// TwinCAT 3 PLC project CPCDAQ_Standard
// ProgramVersion: 3.1.4024.0
// libraries:
//   Tc2_Standard, * (Beckhoff Automation GmbH)
//   Tc2_System, * (Beckhoff Automation GmbH)
//   Tc3_Module, * (Beckhoff Automation GmbH)
// project tree:
//   GVLs/ GVL.TcGVL
//   / PlcTask.TcTTO
//   POUs/ MAIN.TcPOU, POU.TcPOU

CONFIGURATION CPCDAQ_Standard
    RESOURCE PLC ON TwinCAT3
        TASK PlcTask(INTERVAL := T#10ms, PRIORITY := 20);
        PROGRAM MAIN WITH PlcTask : MAIN;
    END_RESOURCE
END_CONFIGURATION

// ---- GVLs/GVL.TcGVL
{attribute 'qualified_only'}
VAR_GLOBAL

(*Digital Input Variables for EL1809 Card*)
bDigital_Input1 AT %I* : BOOL; 
bDigital_Input2 AT %I* : BOOL; 
bDigital_Input3 AT %I* : BOOL; 
bDigital_Input4 AT %I* : BOOL; 
bDigital_Input5 AT %I* : BOOL; 
bDigital_Input6 AT %I* : BOOL; 
bDigital_Input7 AT %I* : BOOL; 
bDigital_Input8 AT %I* : BOOL; 
bDigital_Input9 AT %I* : BOOL; 
bDigital_Input10 AT %I* : BOOL; 
bDigital_Input11 AT %I* : BOOL; 
bDigital_Input12 AT %I* : BOOL; 
bDigital_Input13 AT %I* : BOOL; 
bDigital_Input14 AT %I* : BOOL; 
bDigital_Input15 AT %I* : BOOL; 
bDigital_Input16 AT %I* : BOOL; 


(*4-20mA Analog Input Variables for EL3114 Card*)
nCurrent_Input1 AT %I* : INT; 
nCurrent_Input2 AT %I* : INT; 
nCurrent_Input3 AT %I* : INT; 
nCurrent_Input4 AT %I* : INT; 
nCurrent_Input1_EU AT %I* : REAL; 
nCurrent_Input2_EU AT %I* : REAL; 
nCurrent_Input3_EU AT %I* : REAL; 
nCurrent_Input4_EU AT %I* : REAL; 

(*0-10V Analog Input Variables for EL3104 Card*)
nVoltage_Input1 AT %I* : INT; 
nVoltage_Input2 AT %I* : INT; 
nVoltage_Input3 AT %I* : INT; 
nVoltage_Input4 AT %I* : INT; 
nVoltage_Input1_EU AT %I* : REAL; 
nVoltage_Input2_EU AT %I* : REAL; 
nVoltage_Input3_EU AT %I* : REAL; 
nVoltage_Input4_EU AT %I* : REAL; 


END_VAR

// ---- POUs/MAIN.TcPOU
PROGRAM MAIN
VAR
END_VAR

END_PROGRAM

// ---- POUs/POU.TcPOU
PROGRAM POU
VAR
END_VAR

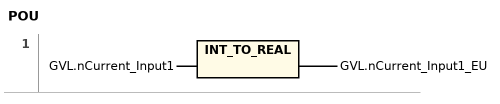
// NETWORK 1
GVL.nCurrent_Input1_EU := INT_TO_REAL(GVL.nCurrent_Input1);

END_PROGRAM
